# B&R Automation Studio project WRAPPER_CTRL
Automation Studio 4.3.11.134 SP; technology packages: mapp 1.63.0

## Configuration Turqueplast

CPU X20CP1382, AutomationRuntime O4.34, Build 4.1.2, Vc V4.34.4

### Hardware
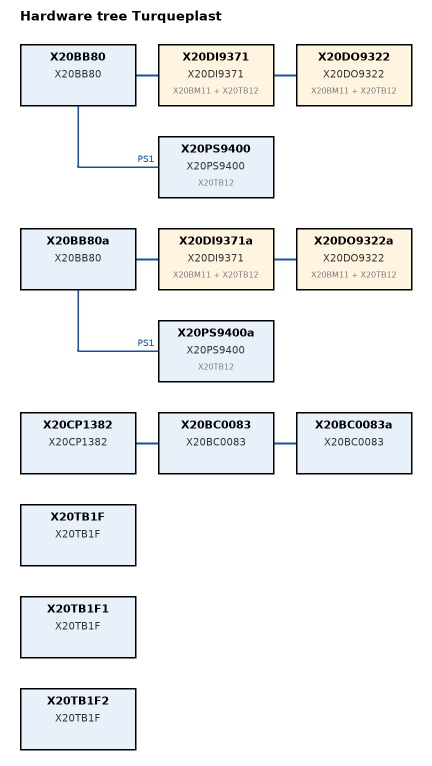
```
X20BB80 : X20BB80 v1.0.2.0
X20BB80a : X20BB80 v1.0.2.0
X20BC0083 : X20BC0083 v2.11.1.0  [PLK1 -> X20CP1382.IF3 (NodeNumber=1) [Cable Type=PowerlinkCable, Length=10, Version=1.0.0.1]; PLK2 -> X20BC0083a.PLK1 (NodeNumber=1) [Cable Type=PowerlinkCable, Length=10, Version=1.0.0.1]; SL -> X20BB80.SL1]
  Supervision = off
X20BC0083a : X20BC0083 v2.11.1.0  [PLK1 -> X20BC0083.PLK2 [Cable Type=PowerlinkCable, Length=10, Version=1.0.0.1]; SL -> X20BB80a.SL1]
  Supervision = off
X20BM11 : X20BM11 v1.0.0.1  [X2X1 -> X20BB80.IF1]
X20BM11a : X20BM11 v1.0.0.1  [X2X1 -> X20BB80a.IF1]
X20BM11b : X20BM11 v1.0.0.1  [X2X1 -> X20BM11.X2X2]
X20BM11c : X20BM11 v1.0.0.1  [X2X1 -> X20BM11a.X2X2]
X20CP1382 : X20CP1382 v1.6.1.0  [X1 -> X1.SL; X2 -> X2.SL; X3 -> X3.SL]
  Module X1 (Type=X1, Virtual=true, Version=1.6.1.0)
    Connection (Connector=SS1, TargetModule=X20TB1F, TargetConnector=SS)
    Connection (Connector=SL, TargetModule=X20CP1382, TargetConnector=X1)
  Module X2 (Type=X2, Virtual=true, Version=1.6.1.0)
    Connection (Connector=SS1, TargetModule=X20TB1F1, TargetConnector=SS)
    Connection (Connector=SL, TargetModule=X20CP1382, TargetConnector=X2)
  Module X3 (Type=X3, Virtual=true, Version=1.6.1.0)
    Connection (Connector=SS1, TargetModule=X20TB1F2, TargetConnector=SS)
    Connection (Connector=SL, TargetModule=X20CP1382, TargetConnector=X3)
  Connector IF2:
    ActivateDevice = 1
    HostName = promass
    Mode = Manual
    InternetAddress = 192.168.3.189  // TURQUEPLAST GIVEN IP
    SubnetMask = 255.255.255.0
  Connector IF3:
    CycleTime = 4000
  ConfigurationID = WRAPPER_CTRL_Turqueplast
  PermanentPvSize = 1000
  RemanentGlobalPvSize = 20000
  EnableUsbRemoteInstall = 1
  EnableCfRemoteInstall = 1
  RebootReset = 1
  Connections = 10
  TimerDeviceType = EPLX2X
  TimerDevice = X20CP1382.IF3
  TaskClassIdleTime = 8000
  Cyclic1Duration = 8000
  Cyclic1Tolerance = 8000
  Cyclic3Duration = 48000
  Cyclic3Tolerance = 48000
  Cyclic8Duration = 8000
  FileDevice1
  FileDeviceName1 = HD
  FileDevicePath1 = C:\RECIPES\
  FileDevice2
  FileDeviceName2 = CF
  FileDevicePath2 = C:\
  FileDevice3
  FileDeviceName3 = LOG
  FileDevicePath3 = C:\LOG\
  EthernetHostName = promass
  EthernetDefaultGateway = 10.0.0.1
  FtpUser1
  FtpUsername1 = bazzica
  FtpUserPassword1 = VS/6Mr2ZWUxRpzYAgWdC7qPbhzWXz9kZH9v1k0AYU+w=
  FtpUserSalt1 = L4/axyh9
  FTPAccessRight1 = 0
  FTPdevice1 = ALL
  FtpUser2
  FtpUsername2 = turque
  FtpUserPassword2 = NA1x5qBXXFgCR/DJGfRfa8Sh4PrFzhFnpgUflhtmUyQ=
  FtpUserSalt2 = yY9t/zs3
  FTPdevice2 = ALL
X20DI9371 : X20DI9371 v1.3.0.0  [SS1 -> X20TB12b.SS; SL -> X20BM11.SL1]
  Supervision = off
X20DI9371a : X20DI9371 v1.3.0.0  [SS1 -> X20TB12c.SS; SL -> X20BM11a.SL1]
  Supervision = off
X20DO9322 : X20DO9322 v1.4.0.0  [SS1 -> X20TB12d.SS; SL -> X20BM11b.SL1]
  Supervision = off
X20DO9322a : X20DO9322 v1.4.0.0  [SS1 -> X20TB12e.SS; SL -> X20BM11c.SL1]
  Supervision = off
X20PS9400 : X20PS9400 v1.3.0.0  [SS1 -> X20TB12.SS; PS -> X20BB80.PS1]
  Supervision = off
X20PS9400a : X20PS9400 v1.3.0.0  [SS1 -> X20TB12a.SS; PS -> X20BB80a.PS1]
  Supervision = off
X20TB12 : X20TB12 v1.0.0.0
X20TB12a : X20TB12 v1.0.0.0
X20TB12b : X20TB12 v1.0.0.0
X20TB12c : X20TB12 v1.0.0.0
X20TB12d : X20TB12 v1.0.0.0
X20TB12e : X20TB12 v1.0.0.0
X20TB1F : X20TB1F v1.0.0.0
X20TB1F1 : X20TB1F v1.0.0.0
X20TB1F2 : X20TB1F v1.0.0.0
```

## Logical view

Binary libraries used (declarations not repeated): operator, runtime, astime, AsIecCon, FileIO, standard

### Global.typ - Global data types
```iecst
TYPE
	typOmronMachine : 	STRUCT
		MCH_on : BOOL;
		Stop : BOOL;
		Run : BOOL;
		NewCycle : BOOL;
		CommitEnd : BOOL;
		Alarm : BOOL;
		AutoMode : BOOL; (*Automatic Mode*)
		ManMode : BOOL; (*Manual Mode*)
		LiveSignal : BOOL; (*Live Signal*)
		LastCycleTime : DINT;
		ActualCycleTime : DINT;
		PcsPerHour : DINT;
		ActualCycleNr : DINT;
		LifeCycles : DINT;
	END_STRUCT;
	typDI : 	STRUCT
		Alarm : BOOL;
		Manual : BOOL;
		Run : BOOL;
		NewCycleSignal : BOOL; (*When Omron Cycle Counter is equal to 1*)
		NewCycleTrigger : BOOL; (*When Omron Cycle Counter is equal to 1*)
		MoldChange : BOOL;
		CommitEnd : BOOL;
	END_STRUCT;
	typAI : 	STRUCT
		DummyAI : REAL;
	END_STRUCT;
	typAO : 	STRUCT
		DummiAO : REAL;
	END_STRUCT;
	typDO : 	STRUCT
		DummyDO : BOOL;
	END_STRUCT;
	typIO : 	STRUCT
		Di : typDI;
		Do : typDO;
		Ai : typAI;
		Ao : typAO;
	END_STRUCT;
	tLocClock : 	STRUCT
		rtcStartUp : DATE_AND_TIME;
		rtcShutDown : DATE_AND_TIME;
		rtcRuntime : DATE_AND_TIME;
		rtcSetTime : DATE_AND_TIME;
		ulTimePlcOff : UDINT;
		myTime : TIME;
	END_STRUCT;
	tCmdClock : 	STRUCT
		bSetClock : BOOL;
		bOkSet : BOOL;
		bErSet : BOOL;
		calSetTime : DTStructure;
	END_STRUCT;
	tGlbClock : 	STRUCT
		alRamData : BOOL;
		alRtcStartUp : BOOL;
		alRtcShutDown : BOOL;
		alRtcRuntime : BOOL;
		rtcRuntime : DATE_AND_TIME;
		calStartUp : DTStructure;
		calShutDown : DTStructure;
		ulTimePlcOff : UDINT;
		cpu_time : UDINT;
		cpu_time_uSec : UDINT;
	END_STRUCT;
END_TYPE
```

### Global.var - Global variables
```iecst
VAR
	M1_NewCycle : TON;
	M2_NewCycle : TON;
	M3_NewCycle : TON;
	gCounter01 : BOOL;
	gCounter02 : BOOL;
	gCounter03 : BOOL;
	gPulse_100 : BOOL;
	gPulse_500 : BOOL;
	gMAC01raw : typIO;
	gMAC02raw : typIO;
	gMAC03raw : typIO;
	gMAC01 : {REDUND_UNREPLICABLE} typOmronMachine := (0);
	gMAC02 : {REDUND_UNREPLICABLE} typOmronMachine := (0);
	gMAC03 : {REDUND_UNREPLICABLE} typOmronMachine := (0);
	gPWL01_ok : BOOL;
	gPWL02_ok : BOOL;
	gPWL03_ok : BOOL;
	cmdClock : tCmdClock;
END_VAR
VAR RETAIN
	glbClock : tGlbClock;
	gMac01CounterOffset : DINT;
	gMac02CounterOffset : DINT;
	gMac03CounterOffset : DINT;
	gMac01LifeCounter : DINT;
	gMac02LifeCounter : DINT;
	gMac03LifeCounter : DINT;
END_VAR
VAR
	glbMac02On : BOOL;
	glbMac01On : BOOL;
END_VAR
```


### Program Logical/main (IEC)

#### Cyclic.ld - Cyclic code
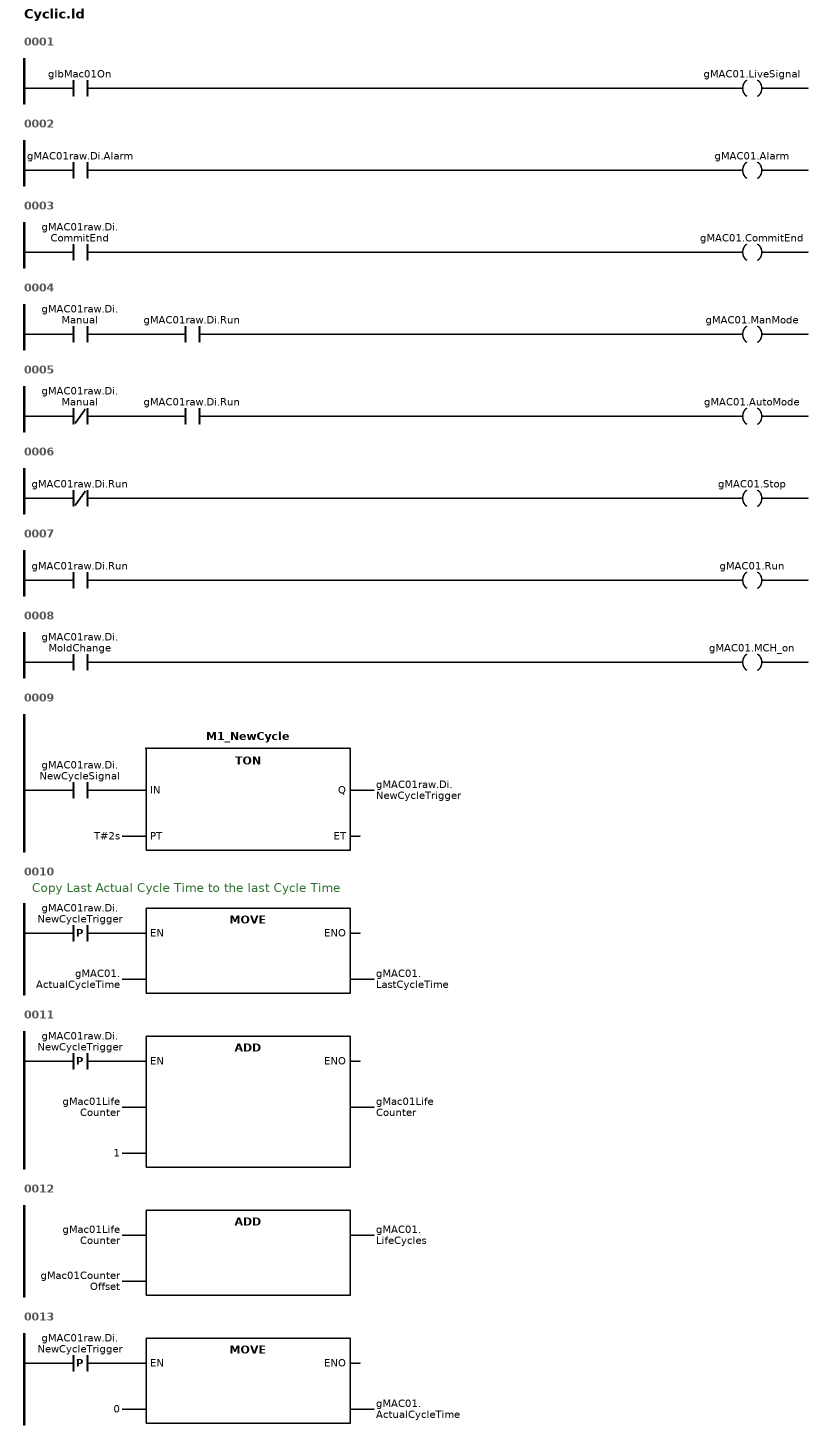
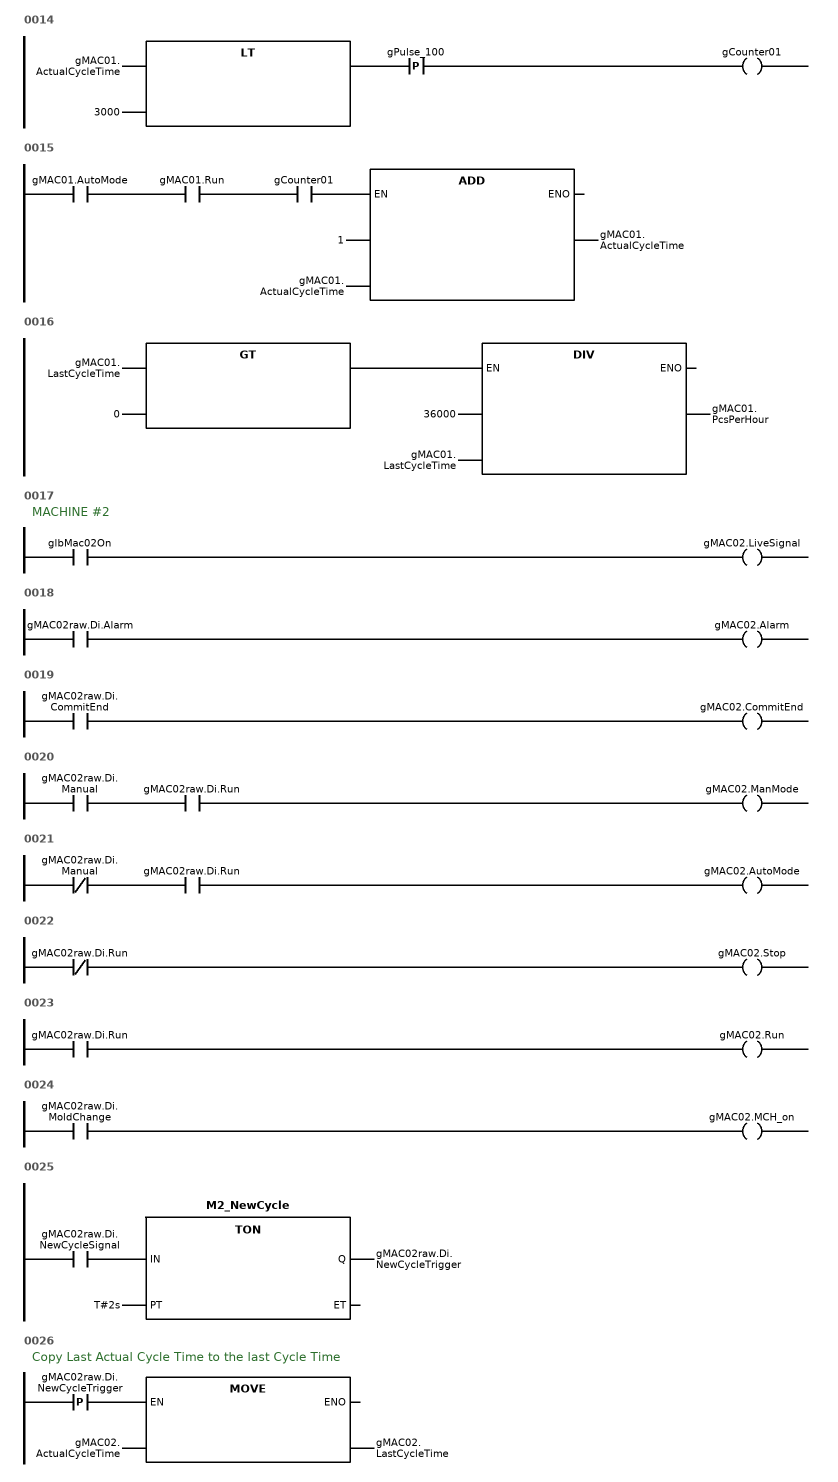
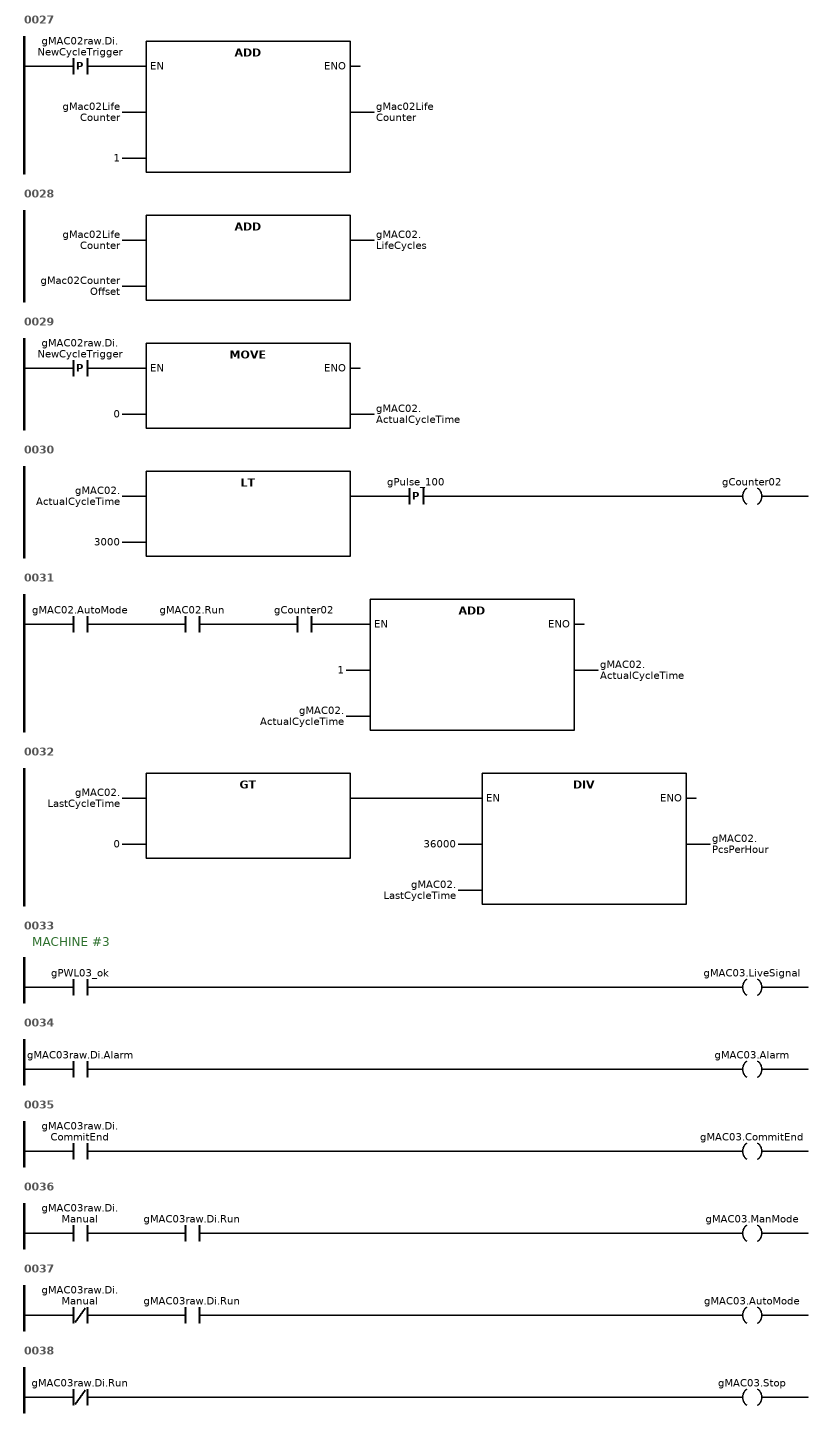
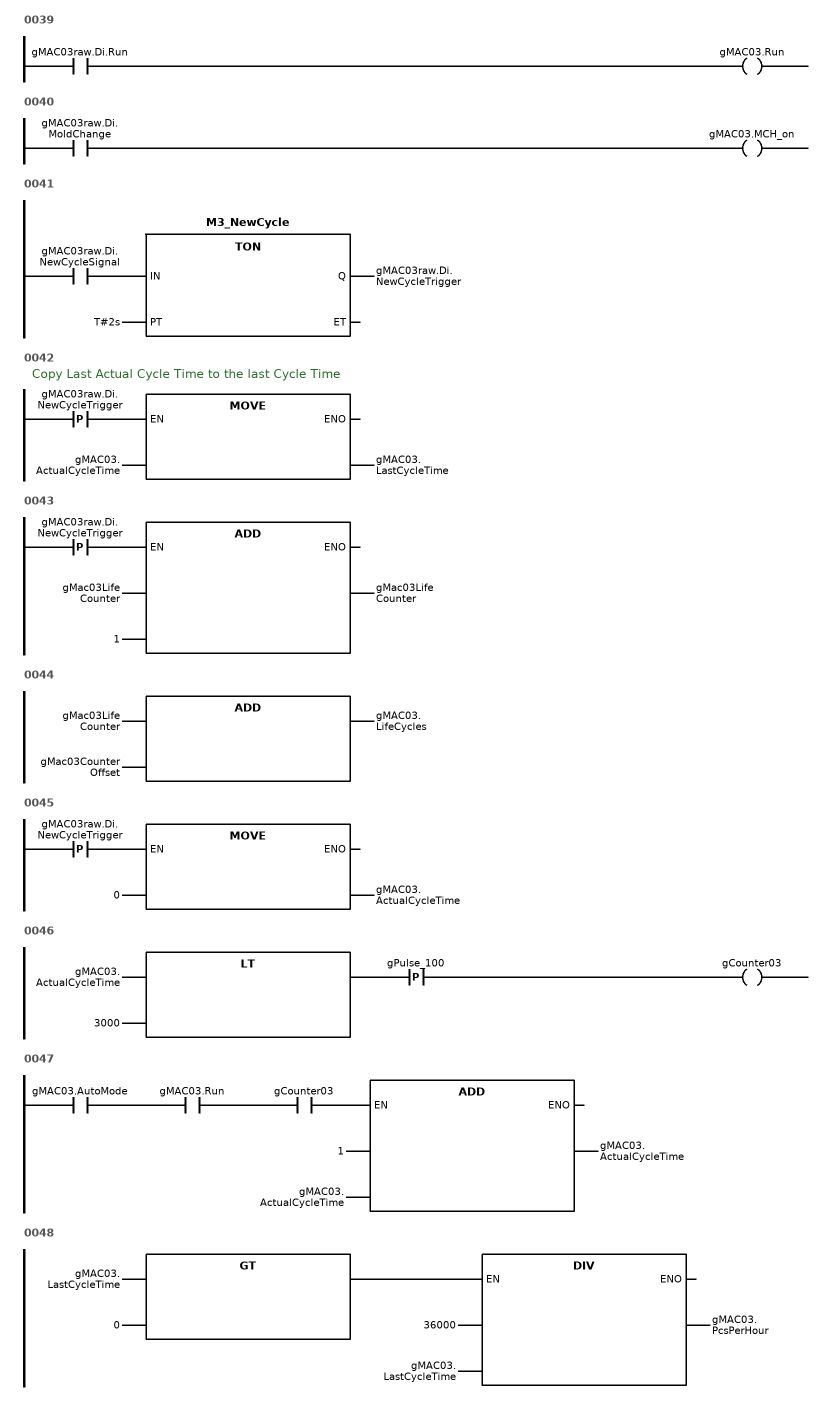
Ladder, written as Structured Text:
```iecst
PROGRAM _CYCLIC
VAR
    _e1 : R_TRIG;
    _e2 : R_TRIG;
    _e3 : R_TRIG;
    _e4 : R_TRIG;
    _p5 : BOOL;
    _p6 : BOOL;
    _e7 : R_TRIG;
    _e8 : R_TRIG;
    _e9 : R_TRIG;
    _e10 : R_TRIG;
    _p11 : BOOL;
    _p12 : BOOL;
    _e13 : R_TRIG;
    _e14 : R_TRIG;
    _e15 : R_TRIG;
    _e16 : R_TRIG;
    _p17 : BOOL;
    _p18 : BOOL;
END_VAR
(* Network 1 *)
gMAC01.LiveSignal := glbMac01On;

(* Network 2 *)
gMAC01.Alarm := gMAC01raw.Di.Alarm;

(* Network 3 *)
gMAC01.CommitEnd := gMAC01raw.Di.CommitEnd;

(* Network 4 *)
gMAC01.ManMode := gMAC01raw.Di.Manual AND gMAC01raw.Di.Run;

(* Network 5 *)
gMAC01.AutoMode := NOT gMAC01raw.Di.Manual AND gMAC01raw.Di.Run;

(* Network 6 *)
gMAC01.Stop := NOT gMAC01raw.Di.Run;

(* Network 7 *)
gMAC01.Run := gMAC01raw.Di.Run;

(* Network 8 *)
gMAC01.MCH_on := gMAC01raw.Di.MoldChange;

(* Network 9 *)
M1_NewCycle(IN := gMAC01raw.Di.NewCycleSignal, PT := T#2s);
gMAC01raw.Di.NewCycleTrigger := M1_NewCycle.Q;

(* Network 10: Copy Last Actual Cycle Time to the last Cycle Time *)
_e1(CLK := gMAC01raw.Di.NewCycleTrigger);
IF _e1.Q THEN gMAC01.LastCycleTime := gMAC01.ActualCycleTime; END_IF;

(* Network 11 *)
_e2(CLK := gMAC01raw.Di.NewCycleTrigger);
IF _e2.Q THEN gMac01LifeCounter := gMac01LifeCounter + 1; END_IF;

(* Network 12 *)
gMAC01.LifeCycles := gMac01LifeCounter + gMac01CounterOffset;

(* Network 13 *)
_e3(CLK := gMAC01raw.Di.NewCycleTrigger);
IF _e3.Q THEN gMAC01.ActualCycleTime := 0; END_IF;

(* Network 14 *)
_e4(CLK := gPulse_100);
gCounter01 := (gMAC01.ActualCycleTime < 3000) AND _e4.Q;

(* Network 15 *)
_p5 := gMAC01.AutoMode AND gMAC01.Run AND gCounter01;
IF _p5 THEN gMAC01.ActualCycleTime := 1 + gMAC01.ActualCycleTime; END_IF;

(* Network 16 *)
_p6 := gMAC01.LastCycleTime > 0;
IF _p6 THEN gMAC01.PcsPerHour := 36000 / gMAC01.LastCycleTime; END_IF;

(* Network 17: MACHINE #2 *)
gMAC02.LiveSignal := glbMac02On;

(* Network 18 *)
gMAC02.Alarm := gMAC02raw.Di.Alarm;

(* Network 19 *)
gMAC02.CommitEnd := gMAC02raw.Di.CommitEnd;

(* Network 20 *)
gMAC02.ManMode := gMAC02raw.Di.Manual AND gMAC02raw.Di.Run;

(* Network 21 *)
gMAC02.AutoMode := NOT gMAC02raw.Di.Manual AND gMAC02raw.Di.Run;

(* Network 22 *)
gMAC02.Stop := NOT gMAC02raw.Di.Run;

(* Network 23 *)
gMAC02.Run := gMAC02raw.Di.Run;

(* Network 24 *)
gMAC02.MCH_on := gMAC02raw.Di.MoldChange;

(* Network 25 *)
M2_NewCycle(IN := gMAC02raw.Di.NewCycleSignal, PT := T#2s);
gMAC02raw.Di.NewCycleTrigger := M2_NewCycle.Q;

(* Network 26: Copy Last Actual Cycle Time to the last Cycle Time *)
_e7(CLK := gMAC02raw.Di.NewCycleTrigger);
IF _e7.Q THEN gMAC02.LastCycleTime := gMAC02.ActualCycleTime; END_IF;

(* Network 27 *)
_e8(CLK := gMAC02raw.Di.NewCycleTrigger);
IF _e8.Q THEN gMac02LifeCounter := gMac02LifeCounter + 1; END_IF;

(* Network 28 *)
gMAC02.LifeCycles := gMac02LifeCounter + gMac02CounterOffset;

(* Network 29 *)
_e9(CLK := gMAC02raw.Di.NewCycleTrigger);
IF _e9.Q THEN gMAC02.ActualCycleTime := 0; END_IF;

(* Network 30 *)
_e10(CLK := gPulse_100);
gCounter02 := (gMAC02.ActualCycleTime < 3000) AND _e10.Q;

(* Network 31 *)
_p11 := gMAC02.AutoMode AND gMAC02.Run AND gCounter02;
IF _p11 THEN gMAC02.ActualCycleTime := 1 + gMAC02.ActualCycleTime; END_IF;

(* Network 32 *)
_p12 := gMAC02.LastCycleTime > 0;
IF _p12 THEN gMAC02.PcsPerHour := 36000 / gMAC02.LastCycleTime; END_IF;

(* Network 33: MACHINE #3 *)
gMAC03.LiveSignal := gPWL03_ok;

(* Network 34 *)
gMAC03.Alarm := gMAC03raw.Di.Alarm;

(* Network 35 *)
gMAC03.CommitEnd := gMAC03raw.Di.CommitEnd;

(* Network 36 *)
gMAC03.ManMode := gMAC03raw.Di.Manual AND gMAC03raw.Di.Run;

(* Network 37 *)
gMAC03.AutoMode := NOT gMAC03raw.Di.Manual AND gMAC03raw.Di.Run;

(* Network 38 *)
gMAC03.Stop := NOT gMAC03raw.Di.Run;

(* Network 39 *)
gMAC03.Run := gMAC03raw.Di.Run;

(* Network 40 *)
gMAC03.MCH_on := gMAC03raw.Di.MoldChange;

(* Network 41 *)
M3_NewCycle(IN := gMAC03raw.Di.NewCycleSignal, PT := T#2s);
gMAC03raw.Di.NewCycleTrigger := M3_NewCycle.Q;

(* Network 42: Copy Last Actual Cycle Time to the last Cycle Time *)
_e13(CLK := gMAC03raw.Di.NewCycleTrigger);
IF _e13.Q THEN gMAC03.LastCycleTime := gMAC03.ActualCycleTime; END_IF;

(* Network 43 *)
_e14(CLK := gMAC03raw.Di.NewCycleTrigger);
IF _e14.Q THEN gMac03LifeCounter := gMac03LifeCounter + 1; END_IF;

(* Network 44 *)
gMAC03.LifeCycles := gMac03LifeCounter + gMac03CounterOffset;

(* Network 45 *)
_e15(CLK := gMAC03raw.Di.NewCycleTrigger);
IF _e15.Q THEN gMAC03.ActualCycleTime := 0; END_IF;

(* Network 46 *)
_e16(CLK := gPulse_100);
gCounter03 := (gMAC03.ActualCycleTime < 3000) AND _e16.Q;

(* Network 47 *)
_p17 := gMAC03.AutoMode AND gMAC03.Run AND gCounter03;
IF _p17 THEN gMAC03.ActualCycleTime := 1 + gMAC03.ActualCycleTime; END_IF;

(* Network 48 *)
_p18 := gMAC03.LastCycleTime > 0;
IF _p18 THEN gMAC03.PcsPerHour := 36000 / gMAC03.LastCycleTime; END_IF;
END_PROGRAM
```

- Program Logical/clock (ANSIC, version 0.00.0) (no source held here)

- Program Logical/Varie (ANSIC) (no source held here)

Listed in the project but not available here: Logical/main/Init.ld, Logical/main/Exit.ld, Logical/main/Types.typ, Logical/main/Variables.var, Logical/clock/clock.var, Logical/clock/clock.c, Logical/Varie/Cyclic.c, Logical/Varie/Init.c, Logical/Varie/Exit.c, Logical/Varie/Types.typ, Logical/Varie/Variables.var
